(* IEC 61131-3 sources: ATCMcontrol_Engineering/src/COM/softing/fc/CL/Libs/ATCM_System, 28 files *)

(* ---- ClearLocalTaskErrno.st ---- *)
(*[[
    UserURL= "ATCMFile:ClearLocalTaskErrno.htm"
]]*)
(*
 *  ATCMControl Standard Function ClearLocalTaskErrno
 *  Purpose: Clears the error state of the given task.
 *)
FUNCTION ClearLocalTaskErrno
VAR_INPUT
    NAME : ANY_STRING;
END_VAR

overload (STRING)  inline {(* add target specific implementaion here *)}
overload (WSTRING) inline {(* add target specific implementaion here *)}

END_FUNCTION

(* ---- ClearTaskErrno.st ---- *)
(*[[
    UserURL= "ATCMFile:ClearTaskErrno.htm"
]]*)
(*
 *  ATCMControl Standard Function ClearTaskErrno
 *  Purpose: Clears the error state variable of the
 *           calling task. Error numbers <>0 signal an
 *           error.
 *)
FUNCTION ClearTaskErrno

;(* add target specific implementaion here *)

END_FUNCTION

(* ---- ColdStartInstance.st ---- *)
(*[[
    UserURL= "ATCMFile:ColdStartInstance.htm"
]]*)
(*
 * ATCMControl standard function ColdStartInstance
 * ----------------------------------------------------------------------------
 * PURPOSE: initialises all program, function block or structure instance members
 *          to their coldstart initial values. This includes also all nested
 *          function blocks and structs.
 *          The function returns if the initialisation is complete.
 *
 * EXAMPLE: StopLocalTask("Task1");
 *          ColdStartInstance("Prog1.myFB");
 *
 * NOTE:    It is recommended to stop the task(s) that operates on "Prog1.myFB"
 *          before calling ColdStartInstance.
 *
 * WARNING: use this function only rarely, it may take a long time to coldstart a
 *          huge and deeply nested instance, that could cause watchdog error in the
 *          calling task. Typically this function is used in a task that also
 *          starts/stops other Tasks and therefore SetSystemTask() was called to
 *          disable the watchdog anyway.
 *)
FUNCTION ColdStartInstance
VAR_INPUT
    instPath : WSTRING;
END_VAR

;(* add target specific implementaion here *)

END_FUNCTION

(* ---- DebugBreak.st ---- *)
(*[[
    UserURL= "ATCMFile:DebugBreak.htm"
]]*)
(*
 *  ATCMControl Standard Function DebugBreak
 *  Purpose: break into the debugger (only if one is attached)
 *)
FUNCTION DebugBreak
VAR_INPUT
    IN : BOOL; (* break only if IN = TRUE *)
END_VAR

;(* add target specific implementaion here *)

END_FUNCTION

(* ---- EnableTaskStatistic.st ---- *)
(*[[
    UserURL= "ATCMFile:EnableTaskStatistic.htm"
]]*)
(*
 *  ATCMControl Standard Function EnableTaskStatistic
 *  Purpose: Enable/Disable the automatic task
 *  statistic output of all tasks.
 *  The default after a download or coldstart or
 *  warmstart is enable=true.
 *
 *  EnableTaskStatistic(true) : enable  task statistics
 *  EnableTaskStatistic(false): disable task statistics
 *)
FUNCTION EnableTaskStatistic
VAR_INPUT
    ENABLE     : BOOL;  (* enable/disable input *)
END_VAR

;(* add target specific implementaion here *)

END_FUNCTION

(* ---- GetComputerName.st ---- *)
(*[[
    UserURL= "ATCMFile:GetComputerName.htm"
]]*)
(*
    Purpose: Gets the computername of the local PC.
*)
FUNCTION GetComputerName : WSTRING

    ;(* add target specific implementaion here *)
    GetComputerName := "?";

END_FUNCTION

(* ---- getCurrentDateAndTime.st ---- *)
(*[[
    UserURL= "ATCMFile:getCurrentDateAndTime.htm"
]]*)

FUNCTION getCurrentDateAndTime : DT

;(* add target specific implementaion here *)
getCurrentDateAndTime := FC_INVALID_DT;

END_FUNCTION

(* ---- GetLocalTaskErrno.st ---- *)
(*[[
    UserURL= "ATCMFile:GetLocalTaskErrno.htm"
]]*)
(*
 *  ATCMControl Standard Function GetLocalTaskErrno
 *  Purpose: get the task error number of the named task.
 *           Return values <>0 signal an error.
 *           See also the FC_ERRNO_* values
 *           defined in ATCM_System.cst.
 *)
FUNCTION GetLocalTaskErrno : DINT
VAR_INPUT
    NAME : ANY_STRING;
END_VAR

overload (STRING)  inline {(* add target specific implementaion here *)}
overload (WSTRING) inline {(* add target specific implementaion here *)}

END_FUNCTION

(* ---- GetLocalTaskState.st ---- *)
(*[[
    UserURL= "ATCMFile:GetLocalTaskState.htm"
]]*)
(*
 *  ATCMControl Standard Function GetLocalTaskState
 *  Purpose: get the current task execution state of the named task.
 *
 *  Possible return values are (see system.cst):
 *  CONST
 *     FC_TASK_STATE_ERROR       : DINT :=-1;
 *     FC_TASK_STATE_ONCREATION  : DINT := 0;
 *     FC_TASK_STATE_STOPPED     : DINT := 1;
 *     FC_TASK_STATE_RUNNING     : DINT := 2;
 *     FC_TASK_STATE_BREAK       : DINT := 3;
 *  END_CONST
 *)
FUNCTION GetLocalTaskState : DINT
VAR_INPUT
    NAME : ANY_STRING;
END_VAR

overload (STRING)  inline {(* add target specific implementaion here *)}
overload (WSTRING) inline {(* add target specific implementaion here *)}

END_FUNCTION

(* ---- GetTaskErrno.st ---- *)
(*[[
    UserURL= "ATCMFile:GetTaskErrno.htm"
]]*)
(*
 *  ATCMControl Standard Function GetTaskErrno
 *  Purpose: returns the last error number of the
 *           calling task.
 *           Return values <>0 signal an error.
 *           See also the FC_ERRNO_* values
 *           defined in 4C_System.cst.
 *)
FUNCTION GetTaskErrno : DINT

;(* add target specific implementaion here *)
GetTaskErrno := 0;

END_FUNCTION

(* ---- getTimeSinceSystemBoot.st ---- *)
(*[[
    UserURL= "ATCMFile:getTimeSinceSystemBoot.htm"
]]*)

FUNCTION getTimeSinceSystemBoot : TIME

;(* add target specific implementaion here *)
getTimeSinceSystemBoot := t#0ms;

END_FUNCTION

(* ---- OutputDebugString.st ---- *)
(*[[
    UserURL= "ATCMFile:OutputDebugString.htm"
]]*)
(*
 *  ATCMControl Standard Functionblock OutputDebugString
 *  Purpose: Write a string to the control's standard output
 *           and the log file. A new line character is added
 *           automatically.
 *)
FUNCTION OutputDebugString
VAR_INPUT
    STR        : ANY_STRING;     (* a one-line message to the user*)
END_VAR

overload (STRING) inline{(* add target specific implementaion here *)}
overload (WSTRING) inline{(* add target specific implementaion here *)}

END_FUNCTION

(* ---- ReadControlVarBOOL.st ---- *)
(*[[
    UserURL= "ATCMFile:ReadControlVarXXXX.htm"
]]*)
(*
 * ATCMControl standard function ReadControlVarBOOL
 * ----------------------------------------------------------------------------
 * PURPOSE: read from a named control variable.
 *
 * EXAMPLE: bValue := ReadControlVarBOOL("Prog1.myFB.aBool");
 *
 * RETURN:  if the function fails, a corresponding
 *          OutputDebugString is made and return is FALSE.
 *
 * WARNING: use this function only rarely, it is not efficient.
 *)
FUNCTION ReadControlVarBOOL : BOOL
VAR_INPUT
   sPath : WSTRING;     (* full qualified name of the variable to read *)
END_VAR

    ;(* add target specific implementaion here *)
    ReadControlVarBOOL := FALSE;
END_FUNCTION

(* ---- ReadControlVarDINT.st ---- *)
(*[[
    UserURL= "ATCMFile:ReadControlVarXXXX.htm"
]]*)
(*
 * ATCMControl standard function ReadControlVarDINT
 * ----------------------------------------------------------------------------
 * PURPOSE: read from a named control variable.
 *
 * EXAMPLE: aInt := ReadControlVarDINT("Prog1.myFB.aInt");
 *
 * RETURN:  if the function fails, a corresponding
 *          OutputDebugString is made and return is 0.
 *
 * WARNING: use this function only rarely, it is not efficient.
 *)
FUNCTION ReadControlVarDINT : DINT
VAR_INPUT
   sPath : WSTRING;     (* full qualified name of the variable to read *)
END_VAR

    ;(* add target specific implementaion here *)
    ReadControlVarDINT := 0;
END_FUNCTION

(* ---- ReadControlVarLINT.st ---- *)
(*[[
    UserURL= "ATCMFile:ReadControlVarXXXX.htm"
]]*)
(*
 * ATCMControl standard function ReadControlVarLINT
 * ----------------------------------------------------------------------------
 * PURPOSE: read from a named control variable.
 *
 * EXAMPLE: aLreal := ReadControlVarLINT("Prog1.myFB.aLint");
 *
 * RETURN:  if the function fails, a corresponding
 *          OutputDebugString is made and return is 0.
 *
 * WARNING: use this function only rarely, it is not efficient.
 *)
FUNCTION ReadControlVarLINT : LINT
VAR_INPUT
   sPath : WSTRING;     (* full qualified name of the variable to read *)
END_VAR

    ;(* add target specific implementaion here *)
    ReadControlVarLINT := 0;

END_FUNCTION

(* ---- ReadControlVarLREAL.st ---- *)
(*[[
    UserURL= "ATCMFile:ReadControlVarXXXX.htm"
]]*)
(*
 * ATCMControl standard function ReadControlVarLREAL
 * ----------------------------------------------------------------------------
 * PURPOSE: read from a named control variable.
 *
 * EXAMPLE: aLreal := ReadControlVarLREAL("Prog1.myFB.aLreal");
 *
 * RETURN:  if the function fails, a corresponding
 *          OutputDebugString is made and return is 0.0.
 *
 * WARNING: use this function only rarely, it is not efficient.
 *)
FUNCTION ReadControlVarLREAL : LREAL
VAR_INPUT
   sPath : WSTRING;     (* full qualified name of the variable to read *)
END_VAR

    ;(* add target specific implementaion here *)
    ReadControlVarLREAL := 0.0;

END_FUNCTION

(* ---- ReadControlVarWSTRING.st ---- *)
(*[[
    UserURL= "ATCMFile:ReadControlVarXXXX.htm"
]]*)
(*
 * ATCMControl standard function ReadControlVarWSTRING
 * ----------------------------------------------------------------------------
 * PURPOSE: read from a named control variable.
 *
 * EXAMPLE: bStr := ReadControlVarWSTRING("Prog1.myFB.aStr");
 *
 * RETURN:  if the function fails, a corresponding
 *          OutputDebugString is made and return is "".
 *
 * WARNING: use this function only rarely, it is not efficient.
 *)
FUNCTION ReadControlVarWSTRING : WSTRING
VAR_INPUT
   sPath : WSTRING;     (* full qualified name of the variable to read *)
END_VAR

    ;(* add target specific implementaion here *)
    ReadControlVarWSTRING  := "";

END_FUNCTION

(* ---- SetSystemTask.st ---- *)
(*[[
    UserURL= "ATCMFile:SetSystemTask.htm"
]]*)
(*
 *  ATCMControl Standard Function SetSystemTask
 *  Purpose: Declare this task to a system task.
 *           To be effective, this has to be the first
 *           statement of the program.
 *           System tasks are tasks that control
 *           other tasks via Start/StopLocalTask.
 *           A System Task will not be checked
 *           for dead-locks, so USE THIS CAREFULLY!
 *)
FUNCTION SetSystemTask

;(* add target specific implementaion here *)

END_FUNCTION

(* ---- SFCResetToInitialStep.st ---- *)
(*[[
    UserURL= "ATCMFile:SFCResetToInitialStep.htm"
]]*)
(*
 *  ATCMControl Standard Function SFCResetToInitialStep
 *  Purpose: reset SFC logic
 *)
FUNCTION SFCResetToInitialStep
VAR_INPUT
    ENABLE : BOOL; (* reset only if ENABLE = TRUE *)
END_VAR

;(* add target specific implementaion here *)

END_FUNCTION

(* ---- StartLocalTask.st ---- *)
(*[[
    UserURL= "ATCMFile:StartLocalTask.htm"
]]*)
(*
 *  ATCMControl Standard Function StartLocalTask
 *  Purpose: Put the named task to the running state.
 *)
FUNCTION StartLocalTask
VAR_INPUT
    NAME : ANY_STRING;
END_VAR

overload (STRING)  inline {(* add target specific implementaion here *)}
overload (WSTRING) inline {(* add target specific implementaion here *)}

END_FUNCTION

(* ---- StopLocalTask.st ---- *)
(*[[
    UserURL= "ATCMFile:StopLocalTask.htm"
]]*)
(*
 *  ATCMControl Standard Function StopLocalTask
 *  Purpose: Put the named task to the stopped state.
 *  WARNING: never try to stop the own task.
 *)
FUNCTION StopLocalTask
VAR_INPUT
    NAME : ANY_STRING;
END_VAR

overload (STRING)  inline {(* add target specific implementaion here *)}
overload (WSTRING) inline {(* add target specific implementaion here *)}

END_FUNCTION

(* ---- WriteControlVarBOOL.st ---- *)
(*[[
    UserURL= "ATCMFile:WriteControlVarXXXX.htm"
]]*)
(*
 * ATCMControl standard function WriteControlVarBOOL
 * ----------------------------------------------------------------------------
 * PURPOSE: write to a named control variable.
 *
 * EXAMPLE: bOk := WriteControlVarBOOL("Prog1.myFB.aBool", TRUE);
 *
 * RETURN:  if the function fails, a corresponding
 *          OutputDebugString is made and return is FALSE.
 *          If successfull the return value is TRUE.
 *
 * WARNING: use this function only rarely, it is not efficient.
 *)
FUNCTION WriteControlVarBOOL : BOOL
VAR_INPUT
   sPath : WSTRING;       (* full qualified name of the variable to write *)
   bVal  : BOOL;          (* value to set *)
END_VAR

    ;(* add target specific implementaion here *)
    WriteControlVarBOOL := FALSE;

END_FUNCTION

(* ---- WriteControlVarDINT.st ---- *)
(*[[
    UserURL= "ATCMFile:WriteControlVarXXXX.htm"
]]*)
(*
 * ATCMControl standard function WriteControlVarDINT
 * ----------------------------------------------------------------------------
 * PURPOSE: write to a named control variable.
 *
 * EXAMPLE: bOk := WriteControlVarDINT("Prog1.myFB.aDint", "42");
 *
 * RETURN:  if the function fails, a corresponding
 *          OutputDebugString is made and return is FALSE.
 *          If successfull the return value is TRUE.
 *
 * WARNING: use this function only rarely, it is not efficient.
 *)
FUNCTION WriteControlVarDINT : BOOL
VAR_INPUT
   sPath : WSTRING;       (* full qualified name of the variable to write *)
   iVal  : DINT;          (* value to set *)
END_VAR

    ;(* add target specific implementaion here *)
    WriteControlVarDINT := FALSE;

END_FUNCTION

(* ---- WriteControlVarLINT.st ---- *)
(*[[
    UserURL= "ATCMFile:WriteControlVarXXXX.htm"
]]*)
(*
 * ATCMControl standard function WriteControlVarLINT
 * ----------------------------------------------------------------------------
 * PURPOSE: write to a named control variable.
 *
 * EXAMPLE: bOk := WriteControlVarLINT("Prog1.myFB.aLint", "42");
 *
 * RETURN:  if the function fails, a corresponding
 *          OutputDebugString is made and return is FALSE.
 *          If successfull the return value is TRUE.
 *
 * WARNING: use this function only rarely, it is not efficient.
 *)
FUNCTION WriteControlVarLINT : BOOL
VAR_INPUT
   sPath : WSTRING;       (* full qualified name of the variable to write *)
   iVal  : LINT;          (* value to set *)
END_VAR

    ;(* add target specific implementaion here *)
    WriteControlVarLINT := FALSE;

END_FUNCTION

(* ---- WriteControlVarLREAL.st ---- *)
(*[[
    UserURL= "ATCMFile:WriteControlVarXXXX.htm"
]]*)
(*
 * ATCMControl standard function WriteControlVarLREAL
 * ----------------------------------------------------------------------------
 * PURPOSE: write to a named control variable.
 *
 * EXAMPLE: bOk := WriteControlVarLREAL("Prog1.myFB.aLreal", "42.0");
 *
 * RETURN:  if the function fails, a corresponding
 *          OutputDebugString is made and return is FALSE.
 *          If successfull the return value is TRUE.
 *
 * WARNING: use this function only rarely, it is not efficient.
 *)
FUNCTION WriteControlVarLREAL : BOOL
VAR_INPUT
   sPath : WSTRING;       (* full qualified name of the variable to write *)
   lVal  : LREAL;         (* value to set *)
END_VAR

    ;(* add target specific implementaion here *)
    WriteControlVarLREAL := FALSE;

END_FUNCTION

(* ---- WriteControlVarWSTRING.st ---- *)
(*[[
    UserURL= "ATCMFile:WriteControlVarXXXX.htm"
]]*)
(*
 * ATCMControl standard function WriteControlVarWSTRING
 * ----------------------------------------------------------------------------
 * PURPOSE: write to a named control variable.
 *
 * EXAMPLE: bOk := WriteControlVarWSTRING("Prog1.myFB.aStr", "hello");
 *
 * RETURN:  if the function fails, a corresponding
 *          OutputDebugString is made and return is FALSE.
 *          If successfull the return value is TRUE.
 *
 * WARNING: use this function only rarely, it is not efficient.
 *)
FUNCTION WriteControlVarWSTRING : BOOL
VAR_INPUT
   sPath : WSTRING;       (* full qualified name of the variable to write *)
   sVal  : WSTRING;       (* value to set *)
END_VAR

    ;(* add target specific implementaion here *)
    WriteControlVarWSTRING  := FALSE;

END_FUNCTION

(* ---- fc_debug.st ---- *)
(*[[
    UserURL= "ATCMFile:FC_DEBUG.htm"
]]*)

(*
 *  ATCMControl Standard Functionblock FC_DEBUG
 *  Purpose: Debug Output
 *)
FUNCTION_BLOCK FC_DEBUG
VAR_INPUT
    ENABLE     : BOOL:=TRUE;  (* enable output with this inst  *)
    STR        : WSTRING;     (* a one-line message to the user*)
END_VAR

IF ENABLE THEN
;(* add target specific implementaion here *)
END_IF;

END_FUNCTION_BLOCK

(* ---- SignalError.st ---- *)
(*[[
    UserURL= "ATCMFile:SignalError.htm"
]]*)
(*
 *  ATCMControl Standard Functionblock SignalError
 *  Purpose: Send Task to Error State
 *
 *  if enable=TRUE and errno<>0 then
 *    the current task is stopped.
 *)
FUNCTION_BLOCK SignalError

VAR_INPUT
    ENABLE     : BOOL:=TRUE;  (* enable this inst *)
    ERRNO      : DINT:=0;     (* error number *)
END_VAR

IF ENABLE AND ERRNO<>0 THEN
;(* add target specific implementaion here *)
END_IF;

END_FUNCTION_BLOCK
